RoboDK station: HAMK_solution_python_kapla_vacuum_gripper_MG400.rdk

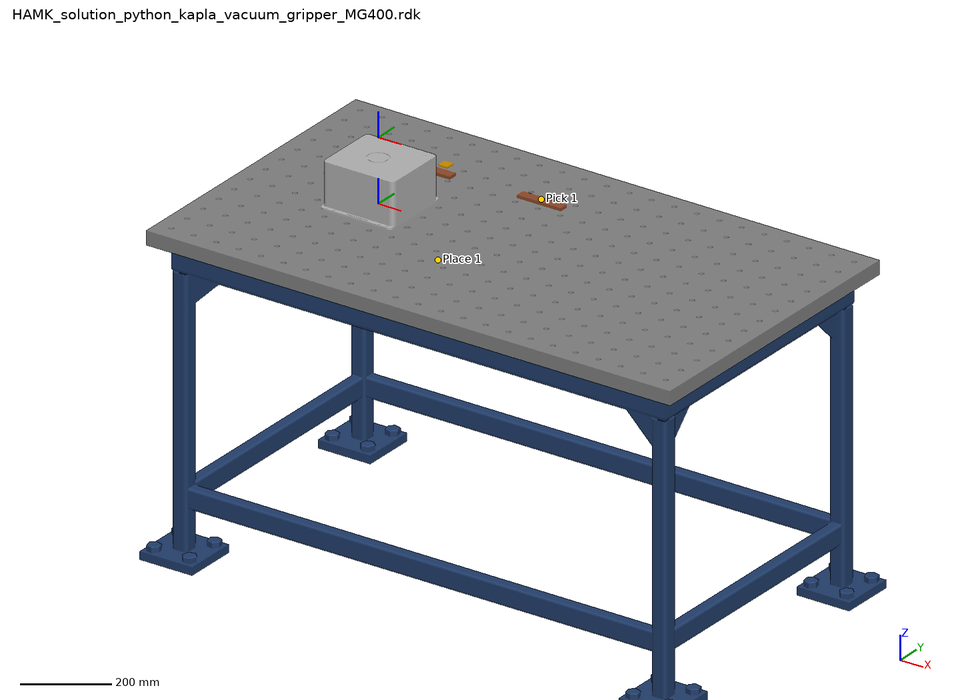
[picture v0: the station drawn from its stored meshes, robots at their saved joint values, targets as dots, program paths as lines]
Station HAMK_solution_python_kapla_vacuum_gripper_MG400 (saved by RoboDK 5.8.0). Poses are relative to the parent item; angles as X-Y-Z fixed-axis rotations.
Station parameters (name, value as stored): IO_1, 1, IO_5, 1, 1, 0, 2, 0
  - frame Dobot MG400 Base at (0, 0, 0) mm
    - robot Dobot MG400: 4 axes, payload 0.5 kg, reach 393.5 mm, repeatability 0.2 mm, weight 4 kg
        joint limits [-160, -25, -25, -360] to [160, 85, 105, 360]; home [0, 0, 0, 0]; saved at [31.827, 70.179, 67.423, 211.827]
      - tool Suction Cup, TCP at (0, 0, -76) mm, size 42.6 x 40 x 76.8 mm
    - frame World at (0, 0, 0) mm
      - object Table at (0, 0, 0) mm, size 1420 x 820 x 800 mm, geometry from Table-1400x800x800mm.sld
        - object HAMK logo at (360, 380, -115) mm, rotated rx 90 ry 0 rz 180 deg, size 301.4 x 100.9 x 9.4 mm, geometry from Fantastic Duup(2).stl
        - object white background at (360, 385.5, -110) mm, rotated rx 90 ry 0 rz 0 deg, size 480 x 184.8 x 2.4 mm, geometry from Fantastic Duup(3).stl
      - object Kapla wood block 0 at (0, 200, 0) mm, size 117 x 23.4 x 7.8 mm, geometry from Kapla wood block.stl
      - object Box at (176, -250, 0) mm, size 76 x 62 x 60 mm, geometry from cube.sld
      - object Mosaic tile 0 at (0, 230, 0) mm, size 24 x 24 x 4 mm, geometry from cube.sld
      - object Mosaic tile 1 at (338.5, -12, 3) mm, size 24 x 24 x 4 mm, geometry from cube.sld
      - object HAMK mosaic frame at (340, -30, 0) mm, size 110 x 100 x 13 mm, geometry from pick_place_frame.stp
      - object Kapla wood block 1 at (290, 210, 0) mm, size 117 x 23.4 x 7.8 mm, geometry from Kapla wood block.stl
  - frame RefSuctionCup at (0, 0, 161.75) mm
    - target Pick 1 (Cartesian target) at (290, 210, -153) mm; joints [35.91, 72.526, 62.197, 215.91] of Dobot MG400
    - target Place 1 (Cartesian target) at (280, -170, -153) mm; joints [-31.264, 68.605, 71.639, 148.736] of Dobot MG400
  - Python program Prog3 (listed below)

--- Python program Prog3 ---
"""
Using Python for pick and place
Fernando Pacheco
2024-12
v4: With wood blocks,
    pick, place and approach positions created programmaticaly
Process:
    Locate Pick 1
    Copy Pick 1
    Loop for i in range(2,num_tiles+1):
        Paste Pick 1 in the reference frame
        Change the name to Pick_i
        Move Pick_i in the y-axis
    Loop for i in range(1,num_tiles+1):
        Paste Pick 1 in the reference frame
        Change the name to Approach_i
        Move Approach_i in the y-axis and z-axis
    Locate Place 1
    Copy Place 1
    Loop for i in range(2,num_tiles+1):
        Paste Place 1 in the reference frame
        Change the name to Place_i
        Translate Place_i in the z-axis and rotate in z-axis

"""

from robodk import robolink    # RoboDK API
from robodk import robomath    # Robot toolbox

from math import radians # to convert degrees to radians

num_tiles=3 # number of mosaic tiles to pick

# Connect to RoboDK
RDK = robolink.Robolink()

# Get the robot
# RDK.Item searches for items in the station
robot = RDK.Item('Dobot MG400', robolink.ITEM_TYPE_ROBOT)

# Get the reference frame
frame = RDK.Item('RefSuctionCup')

# Get the target Pick 1, copy it
pick = RDK.Item('Pick 1')
pick.Copy() # equivalent to using CTRL+C

for i in range(2, num_tiles+1):
    temp = frame.Paste() # equivalent to CTRL+V
    temp.setName('Pick '+str(i))
    temp.setPose(temp.Pose()*robomath.transl(ty=-30*(i-1)))

# similar to Approach_i
for i in range(1, num_tiles+1):
    temp = frame.Paste() # equivalent to CTRL+V
    temp.setName('AppPick '+str(i))
    temp.setPose(temp.Pose()*robomath.transl(ty=-30*(i-1), tz=80))

place = RDK.Item('Place 1')
place.Copy()
for i in range(2, num_tiles+1):
    temp = frame.Paste() # equivalent to CTRL+V
    temp.setName('Place '+str(i))
    temp.setPose(temp.Pose()*robomath.transl(tz=+7.9*(i-1)))
    temp.setPose(temp.Pose()*robomath.rotz(rz=radians(45)*(i-1)))

for i in range(1, num_tiles+1):
    place = RDK.Item('Place '+str(i))
    place.Copy()
    temp = frame.Paste() # equivalent to CTRL+V
    temp.setName('AppPlace '+str(i))
    temp.setPose(temp.Pose()*robomath.transl(tz=+45))

# Movements
for i in range(1, num_tiles+1):
    approach_pick = RDK.Item('AppPick '+str(i))
    approach_place = RDK.Item('AppPlace '+str(i))
    pick = RDK.Item('Pick '+str(i))
    place = RDK.Item('Place '+str(i))
    robot.MoveJ(approach_pick)
    robot.MoveL(pick)
    robot.setDO('1',1) # turn on Vacuum
    robot.Pause(200)
    robot.MoveL(approach_pick)
    robot.MoveJ(approach_place)
    robot.MoveL(place)
    robot.setDO('1',0)
    robot.setDO('2',1) # turn on Pressure
    robot.Pause(200)
    robot.setDO('2',0)
    robot.MoveL(approach_place)
